(* CoDeSys 2.3 export: GVL_WRITE.EXP *)

(* Global variable list: AdsClientTests/GVL_Write *)
VAR_GLOBAL
	Write_StandardTypes 		: ST_StandardTypes;
	Write_StandardArrays 		: ST_StandardArrayTypes;
	Write_ComplexTypes		: ST_ComplexTypes;
	Write_ComplexArrayTypes	: ST_ComplexArrayTypes;
	Write_SpecialTypes		: ST_SpecialTypes;
	Write_IssueSpecificTypes	: ST_IssueSpecificTypes;
END_VAR
